FUNCTION fDegToRad : REAL
VAR_INPUT
	rDegrees		:REAL;
END_VAR
VAR
END_VAR

fDegToRad:=((rDegrees*PI)/180);

END_FUNCTION

(* stored: Version 1.1.0.1, ProductVersion 3.1.4024.12
   POU fDegToRad: Id {dc27d456-5289-4572-b677-fc28a12c224a}, SpecialFunc None *)
